(* IEC 61131-3 sources: Industry-PLC-LLM/data/PLCBEAD_repo/PLCBEAD_PLCEmbed-main/PLC-BEAD/Source/GEB/RES_PT, 1 file *)

(* ---- RES_PT.ST ---- *)
FUNCTION RES_PT:REAL
	VAR_INPUT
		T :	REAL;
		R0 :	REAL;
	END_VAR

	VAR
		T2 :	REAL;
	END_VAR

	T2 := T * T;

	IF T >= 0.0 THEN
		RES_PT := R0 * ( 1.0 + 3.90802E-3 * T + -5.802E-7 * T2);
	ELSE
		RES_PT := R0 * ( 1.0 + 3.90802E-3 * T + -5.802E-7 * T2 + -4.27350E-12 * (T - 100.0) * T2 * T);
	END_IF;

END_FUNCTION

PROGRAM program0
  	VAR
		T :	REAL;
		R0 : REAL;
		CEIL5_OUT : REAL;
  	END_VAR

  	CEIL5_OUT := RES_PT(T, R0);
END_PROGRAM
